(* IEC 61131-3 sources: nvidia-ai-factory-controls/libraries/AIFactory_Common/POUs/Control, 6 files *)

(* ---- FB_AlarmManager.fb ---- *)
(* =============================================================================
    FB_AlarmManager — Alarm Buffer, Acknowledge, History
    Common Library | NVIDIA AI Factory Controls
   =============================================================================

   PURPOSE:
     Manages a circular buffer of 100 alarm records. Provides methods to
     raise, clear, and acknowledge alarms. Tracks active/unacknowledged
     counts and critical alarm presence.

   DESIGN:
     - Circular buffer: oldest alarm overwritten when full
     - Alarm identified by nID (unique per alarm point)
     - Raise = create/activate alarm record with timestamp
     - Clear = mark alarm inactive (condition returned to normal)
     - Acknowledge = mark alarm acknowledged by operator
     - Thread-safe: designed for single-task use

   USAGE:
     Call M_Execute() once per scan (via base class lifecycle).
     Call M_RaiseAlarm() when a condition triggers an alarm.
     Call M_ClearAlarm() when the alarm condition returns to normal.
     Call M_Acknowledge() from HMI/SCADA command handler.

   EXTENDS: FB_Base
   ============================================================================= *)

(* ═══════════════════════════════════════════════════════════════════════════════
   DECLARATION
   ═══════════════════════════════════════════════════════════════════════════════ *)

{attribute 'no_assign'}
FUNCTION_BLOCK FB_AlarmManager EXTENDS FB_Base
VAR_INPUT
    (* ─── Timing ─── *)
    fCycleTime_s         : REAL := 0.005;   (* Task cycle [seconds] *)
END_VAR

VAR_OUTPUT
    (* ─── Summary Status ─── *)
    nActiveCount         : UDINT;           (* Number of currently active alarms *)
    nUnacknowledgedCount : UDINT;           (* Number of unacknowledged alarms *)
    bAnyCritical         : BOOL;            (* TRUE if any CRITICAL alarm is active *)
    nTotalAlarms         : UDINT;           (* Total alarms in buffer *)
END_VAR

VAR
    (* ─── Circular Buffer ─── *)
    _astBuffer           : ARRAY[1..100] OF ST_AlarmRecord;
    _nWriteIndex         : UDINT := 1;     (* Next write position *)
    _nBufferCount        : UDINT := 0;     (* Number of valid entries *)

    (* ─── Edge Triggers for count transitions ─── *)
    _rtrigRaise          : R_TRIG;         (* Rising edge on raise event *)
    _rtrigClear          : R_TRIG;         (* Rising edge on clear event *)

    (* ─── Internal Flags ─── *)
    _bRaiseEvent         : BOOL;           (* Pulse: alarm raised this scan *)
    _bClearEvent         : BOOL;           (* Pulse: alarm cleared this scan *)

    (* ─── Loop Variable ─── *)
    _i                   : UDINT;
END_VAR

VAR CONSTANT
    C_BUFFER_SIZE        : UDINT := 100;
END_VAR

(* ═══════════════════════════════════════════════════════════════════════════════
   IMPLEMENTATION
   ═══════════════════════════════════════════════════════════════════════════════ *)

(* Base class lifecycle handles enable/init/fault/execute gating *)
SUPER^();

(* ---- FB_EdgeDetector.fb ---- *)
(* =============================================================================
    FB_EdgeDetector — Combined Rising/Falling Edge Detection
    Common Library | NVIDIA AI Factory Controls
   =============================================================================

   PURPOSE:
     Convenience wrapper providing BOTH rising and falling edge outputs
     from a single BOOL input. Reduces variable count when you need both.

   WHEN TO USE:
     • State transition logging (need to know WHEN it changed, not just state)
     • Pump start/stop counting (R_TRIG for start, F_TRIG for stop)
     • Alarm event generation (rising = alarm raised, falling = alarm cleared)
     • One-shot command execution (only act on the transition, not the level)

   STANDARD R_TRIG/F_TRIG vs THIS FB:
     Use standard R_TRIG/F_TRIG when you only need one edge direction.
     Use this FB when you need both edges from the same signal.

   USAGE:
     fbPumpEdge(bInput := bDI_PumpRunning);
     IF fbPumpEdge.bRising THEN
         nStartCount := nStartCount + 1;
     END_IF
     IF fbPumpEdge.bFalling THEN
         // Pump stopped unexpectedly — alarm
     END_IF
   ============================================================================= *)

(* ═══════════════════════════════════════════════════════════════════════════════
   DECLARATION
   ═══════════════════════════════════════════════════════════════════════════════ *)

FUNCTION_BLOCK FB_EdgeDetector
VAR_INPUT
    bInput               : BOOL;            (* Signal to monitor *)
END_VAR

VAR_OUTPUT
    bRising              : BOOL;            (* TRUE for one scan on 0→1 transition *)
    bFalling             : BOOL;            (* TRUE for one scan on 1→0 transition *)
    bChanged             : BOOL;            (* TRUE for one scan on ANY change *)
END_VAR

VAR
    _rtrig               : R_TRIG;
    _ftrig               : F_TRIG;
END_VAR

(* ═══════════════════════════════════════════════════════════════════════════════
   IMPLEMENTATION
   ═══════════════════════════════════════════════════════════════════════════════ *)

_rtrig(CLK := bInput);
_ftrig(CLK := bInput);

bRising := _rtrig.Q;
bFalling := _ftrig.Q;
bChanged := bRising OR bFalling;

(* ---- FB_PID.fb ---- *)
(* =============================================================================
    FB_PID — Industrial PID Controller with Safety Features
    Common Library | NVIDIA AI Factory Controls
   =============================================================================

   PURPOSE:
     Production-grade PID controller for process control loops.
     Used by cooling (pump speed, valve position) and power (setpoints).

   FEATURES:
     • Anti-windup via integrator clamping + back-calculation
     • Derivative on PV (avoids setpoint kick)
     • Filtered derivative (noise rejection)
     • Bumpless manual↔auto transfer
     • Output rate limiting (prevents water hammer, VFD stress)
     • Setpoint weighting on P-term
     • Configurable deadband

   SAFETY:
     • Extends FB_Base: inherits enable/fault/safe-state lifecycle
     • Safe-state: output = 0.0 (or configured safe output)
     • Input validation: rejects NaN/Inf setpoints and PV
     • Cycle time validation: rejects zero or negative

   RACE CONDITION PREVENTION:
     • Single-task ownership. Never share across tasks.
     • All parameters are VAR_INPUT (written by owner task only).
     • Output is a single REAL — atomically readable by other tasks
       if needed (but prefer ST_* snapshot pattern).

   TUNING GUIDE:
     Kp = Controller gain (higher = more aggressive)
     Ti = Integral time [s] (lower = faster integral action; 0 = off)
     Td = Derivative time [s] (higher = more damping; 0 = off)
     Start with: Kp=1.0, Ti=60.0, Td=0.0, then tune from there.
   ============================================================================= *)

(* ═══════════════════════════════════════════════════════════════════════════════
   DECLARATION
   ═══════════════════════════════════════════════════════════════════════════════ *)

FUNCTION_BLOCK FB_PID EXTENDS FB_Base
VAR_INPUT
    (* --- Process Variables --- *)
    fSetpoint            : REAL;            (* Desired value [eng. units] *)
    fProcessValue        : REAL;            (* Measured value [eng. units] *)

    (* --- Tuning Parameters --- *)
    fKp                  : REAL := 1.0;     (* Proportional gain *)
    fTi                  : REAL := 60.0;    (* Integral time [s]; 0=disabled *)
    fTd                  : REAL := 0.0;     (* Derivative time [s]; 0=disabled *)
    fDerivFilterN        : REAL := 10.0;    (* Derivative filter coeff (2..20) *)
    fSPWeight            : REAL := 1.0;     (* Setpoint weight for P-term [0..1] *)

    (* --- Output Limits --- *)
    fOutputMin           : REAL := 0.0;     (* Minimum output *)
    fOutputMax           : REAL := 100.0;   (* Maximum output *)
    fRateLimit           : REAL := 0.0;     (* Max output change [units/s]; 0=off *)

    (* --- Deadband --- *)
    fDeadband            : REAL := 0.0;     (* Error deadband [eng. units] *)

    (* --- Manual Mode --- *)
    bManualMode          : BOOL;            (* TRUE = manual output override *)
    fManualOutput        : REAL;            (* Manual output value *)

    (* --- Timing --- *)
    fCycleTime_s         : REAL := 0.005;   (* Task cycle time [seconds] *)

    (* --- Safe Output (used in safe-state) --- *)
    fSafeOutput          : REAL := 0.0;     (* Output value when disabled/faulted *)
END_VAR

VAR_OUTPUT
    (* --- Control Output --- *)
    fOutput              : REAL;            (* Controller output [OutputMin..OutputMax] *)

    (* --- Diagnostics --- *)
    fError               : REAL;            (* Current error: SP - PV *)
    fP_Term              : REAL;            (* Proportional contribution *)
    fI_Term              : REAL;            (* Integral contribution *)
    fD_Term              : REAL;            (* Derivative contribution *)
    bAtUpperLimit        : BOOL;            (* Output clamped at max *)
    bAtLowerLimit        : BOOL;            (* Output clamped at min *)
    bIsManual            : BOOL;            (* Currently in manual mode *)
END_VAR

VAR
    (* --- Internal State --- *)
    _fIntegral           : REAL;            (* Integral accumulator *)
    _fDerivState         : REAL;            (* Derivative filter state *)
    _fPV_Prev            : REAL;            (* Previous PV for derivative *)
    _fOutputPrev         : REAL;            (* Previous output for rate limit *)
    _bWindupHigh         : BOOL;            (* Positive saturation detected *)
    _bWindupLow          : BOOL;            (* Negative saturation detected *)
END_VAR

(* ═══════════════════════════════════════════════════════════════════════════════
   IMPLEMENTATION
   ═══════════════════════════════════════════════════════════════════════════════ *)

(* Lifecycle managed by FB_Base. Actual PID logic in M_Execute. *)
SUPER^();

(* ---- FB_RampGenerator.fb ---- *)
(* =============================================================================
    FB_RampGenerator — Reusable Output Ramping Utility
    Common Library | NVIDIA AI Factory Controls
   =============================================================================

   PURPOSE:
     Provides linear ramping from current output toward a target value
     at a configurable rate. Used for pump speed ramping, valve position
     ramping, and any analog output that requires rate-limiting.

   BEHAVIOR:
     - bEnable=TRUE: ramps fOutput toward fTarget at fRampRate units/second
     - bEnable=FALSE: holds current fOutput (freeze)
     - bReset=TRUE: jumps immediately to fTarget (no ramp)
     - Output always clamped between fMin and fMax
     - bAtTarget=TRUE when fOutput equals fTarget (within float tolerance)

   DESIGN:
     Standalone utility FB — does NOT extend FB_Base.
     Lightweight, composable, no lifecycle overhead.
   ============================================================================= *)

(* ═══════════════════════════════════════════════════════════════════════════════
   DECLARATION
   ═══════════════════════════════════════════════════════════════════════════════ *)

FUNCTION_BLOCK FB_RampGenerator
VAR_INPUT
    fTarget          : REAL;                (* Desired output value [units] *)
    fRampRate        : REAL;                (* Maximum change rate [units/second] *)
    fCycleTime_s     : REAL;                (* Task cycle time [seconds] *)
    bEnable          : BOOL;                (* TRUE = ramp active; FALSE = freeze *)
    bReset           : BOOL;                (* TRUE = jump immediately to target *)
    fMin             : REAL := 0.0;         (* Minimum output clamp [units] *)
    fMax             : REAL := 100.0;       (* Maximum output clamp [units] *)
END_VAR

VAR_OUTPUT
    fOutput          : REAL;                (* Current ramped output value [units] *)
    bAtTarget        : BOOL;                (* TRUE when fOutput = fTarget *)
END_VAR

VAR
    _fMaxStep        : REAL;                (* Max change per scan [units] *)
    _fError          : REAL;                (* Distance to target [units] *)
END_VAR

VAR CONSTANT
    C_TOLERANCE      : REAL := 0.001;       (* At-target deadband [units] *)
END_VAR

(* ═══════════════════════════════════════════════════════════════════════════════
   IMPLEMENTATION
   ═══════════════════════════════════════════════════════════════════════════════ *)

(* ─── Reset: immediate jump to target ────────────────────────────────────────── *)
IF bReset THEN
    fOutput := fTarget;
END_IF

(* ─── Ramp logic (only when enabled and not reset) ───────────────────────────── *)
IF bEnable AND NOT bReset THEN
    (* Calculate maximum step per scan *)
    _fMaxStep := fRampRate * fCycleTime_s;

    (* Calculate distance to target *)
    _fError := fTarget - fOutput;

    (* Apply rate-limited step *)
    IF ABS(_fError) <= _fMaxStep THEN
        (* Close enough — snap to target *)
        fOutput := fTarget;
    ELSIF _fError > 0.0 THEN
        (* Ramp up *)
        fOutput := fOutput + _fMaxStep;
    ELSE
        (* Ramp down *)
        fOutput := fOutput - _fMaxStep;
    END_IF
END_IF

(* ─── Clamp output to configured limits ──────────────────────────────────────── *)
IF fOutput < fMin THEN
    fOutput := fMin;
ELSIF fOutput > fMax THEN
    fOutput := fMax;
END_IF

(* ─── At-target detection ────────────────────────────────────────────────────── *)
bAtTarget := (ABS(fOutput - fTarget) <= C_TOLERANCE);

(* ---- FB_SensorValidator.fb ---- *)
(* =============================================================================
    FB_SensorValidator — Input Signal Validation & Filtering
    Common Library | NVIDIA AI Factory Controls
   =============================================================================

   PURPOSE:
     Validates raw analog sensor inputs before they reach control logic.
     Implements defense-in-depth for sensor data:
       1. Range check (physical limits)
       2. Rate-of-change check (spike/noise rejection)
       3. Redundancy voting (if dual sensors available)
       4. First-order low-pass filtering
       5. Stale-data detection (frozen signal)

   SAFETY PRINCIPLE:
     Control logic NEVER reads raw I/O directly. Every sensor passes
     through this FB. If validation fails, output.bValid = FALSE and
     output.fValue = configured fallback (safe value).

   RACE CONDITION PREVENTION:
     • One instance per sensor, owned by one task.
     • Output struct (ST_SensorInput) is copied atomically to shared memory
       by the owning task — never written field-by-field across tasks.

   USAGE:
     fbTempSensor(
         fRawInput := IO_Module.AI_Temperature,
         stConfig  := stTempSensorConfig
     );
     // Use fbTempSensor.stOutput.fValue only if fbTempSensor.stOutput.bValid
   ============================================================================= *)

(* ═══════════════════════════════════════════════════════════════════════════════
   DECLARATION
   ═══════════════════════════════════════════════════════════════════════════════ *)

FUNCTION_BLOCK FB_SensorValidator EXTENDS FB_Base
VAR_INPUT
    fRawInput            : REAL;            (* Raw analog value from I/O module *)
    fRawInput_Redundant  : REAL;            (* Redundant sensor (0.0 if unused) *)
    bUseRedundancy       : BOOL;            (* TRUE = dual-sensor voting active *)
    fCycleTime_s         : REAL := 0.005;   (* Task cycle time [seconds] *)

    (* --- Configuration (typically set once at startup) --- *)
    fRangeLow            : REAL := 0.0;     (* Physical minimum [eng. units] *)
    fRangeHigh           : REAL := 100.0;   (* Physical maximum [eng. units] *)
    fMaxRateOfChange     : REAL := 50.0;    (* Max valid rate [units/s]; 0=off *)
    fRedundancyTolerance : REAL := 2.0;     (* Max diff between sensors [units] *)
    fFilterTimeConst     : REAL := 0.5;     (* Low-pass filter tau [seconds] *)
    fFallbackValue       : REAL := 0.0;     (* Value when invalid *)
    fFrozenTimeout_s     : REAL := 30.0;    (* Frozen signal timeout [seconds] *)
    sTag                 : STRING(32) := 'UNNAMED'; (* Sensor tag for diagnostics *)
END_VAR

VAR_OUTPUT
    stOutput             : ST_SensorInput;  (* Validated output structure *)
    bAlm_OutOfRange      : BOOL;            (* Value outside physical limits *)
    bAlm_RateExceeded    : BOOL;            (* Spike/noise detected *)
    bAlm_RedundancyFault : BOOL;            (* Dual sensors disagree *)
    bAlm_Frozen          : BOOL;            (* Signal not changing (stuck) *)
END_VAR

VAR
    _fPrevValue          : REAL;            (* Previous scan value for rate calc *)
    _fFiltered           : REAL;            (* Filtered output *)
    _fFilterAlpha        : REAL;            (* Computed filter coefficient *)
    _fFrozenTimer_s      : REAL;            (* Accumulates time signal unchanged *)
    _fFrozenLastValue    : REAL;            (* Last value that was different *)
    _nFaultCount         : UINT;            (* Consecutive fault counter *)
    _nMaxFaultCount      : UINT := 10;      (* Faults before declaring invalid *)
    _bFirstScan          : BOOL := TRUE;    (* First-scan initialization flag *)
END_VAR

(* ═══════════════════════════════════════════════════════════════════════════════
   IMPLEMENTATION
   ═══════════════════════════════════════════════════════════════════════════════ *)

(* Call base class — handles lifecycle, heartbeat, enable/fault gates *)
SUPER^();

(* NOTE: Actual sensor logic is in M_Execute override below.
   This body only calls the base class. All work is in the virtual methods. *)

(* ---- FB_Watchdog.fb ---- *)
(* =============================================================================
    FB_Watchdog — External Watchdog Kick/Monitor
    Common Library | NVIDIA AI Factory Controls
   =============================================================================

   PURPOSE:
     Monitors an external heartbeat counter from another task or IPC.
     Detects if the heartbeat stops incrementing (stale) and reports
     a timeout condition.

   BEHAVIOR:
     - Compares current nExternalHeartbeat with stored previous value
     - If changed: resets timeout accumulator, bAlive=TRUE
     - If unchanged: accumulates time, triggers bTimeout after nTimeout_ms
     - R_TRIG on bTimeout transition for one-shot fault notification

   USE CASES:
     - Control_Task monitoring Safety_Task heartbeat
     - Edge gateway monitoring IPC application heartbeat
     - Any cross-task/cross-IPC liveness check

   DESIGN:
     Simple utility FB — does NOT extend FB_Base.
     Lightweight, composable, no lifecycle overhead.
   ============================================================================= *)

(* ═══════════════════════════════════════════════════════════════════════════════
   DECLARATION
   ═══════════════════════════════════════════════════════════════════════════════ *)

FUNCTION_BLOCK FB_Watchdog
VAR_INPUT
    nExternalHeartbeat   : UDINT;           (* External heartbeat counter to monitor *)
    nTimeout_ms          : UDINT := 1000;   (* Max time without change [ms] *)
    fCycleTime_s         : REAL := 0.005;   (* This task's cycle time [seconds] *)
END_VAR

VAR_OUTPUT
    bAlive               : BOOL;            (* TRUE if heartbeat is changing *)
    bTimeout             : BOOL;            (* TRUE if heartbeat stale beyond timeout *)
END_VAR

VAR
    _nPrevHeartbeat      : UDINT;           (* Previous scan's heartbeat value *)
    _fTimeSinceChange    : REAL;            (* Accumulated time since last change [s] *)
    _fTimeout_s          : REAL;            (* Timeout converted to seconds *)
    _rtrigTimeout        : R_TRIG;          (* Rising edge on timeout for one-shot *)
    _bFirstScan          : BOOL := TRUE;    (* Guards first-scan initialization *)
END_VAR

(* ═══════════════════════════════════════════════════════════════════════════════
   IMPLEMENTATION
   ═══════════════════════════════════════════════════════════════════════════════ *)

(* ─── First scan: initialize previous value ──────────────────────────────────── *)
IF _bFirstScan THEN
    _nPrevHeartbeat := nExternalHeartbeat;
    _fTimeSinceChange := 0.0;
    _bFirstScan := FALSE;
END_IF

(* ─── Convert timeout to seconds ─────────────────────────────────────────────── *)
_fTimeout_s := UDINT_TO_REAL(nTimeout_ms) / 1000.0;

(* ─── Compare heartbeat with previous value ───────────────────────────────────── *)
IF nExternalHeartbeat <> _nPrevHeartbeat THEN
    (* Heartbeat changed — external task is alive *)
    _fTimeSinceChange := 0.0;
    bAlive := TRUE;
    bTimeout := FALSE;
    _nPrevHeartbeat := nExternalHeartbeat;
ELSE
    (* Heartbeat unchanged — accumulate time *)
    _fTimeSinceChange := _fTimeSinceChange + fCycleTime_s;

    (* Check timeout *)
    IF _fTimeSinceChange >= _fTimeout_s THEN
        bAlive := FALSE;
        bTimeout := TRUE;
    END_IF
END_IF

(* ─── R_TRIG for one-shot timeout notification ───────────────────────────────── *)
_rtrigTimeout(CLK := bTimeout);
